Fanuc KAREL source: kt00452.KL

-- PROVISIONAL review KL for V770-1; original PC SHA256 5246766105a77e096c1f6754eb6137f0ccf5cd3cca0d1063bb0bf1915763c5d0
-- Incomplete behavior may be omitted. Consult companion uncertainty JSON. Do not deploy.
PROGRAM KT00452
%NOLOCKGROUP
VAR
  R2 : REAL
  OUT : BOOLEAN
-- UNRESOLVED_DECL H1 type=002017
BEGIN
  -- UNRESOLVED_PC offsets 5-19; opcodes 2E,22,9D,33,B4
  -- UNRESOLVED_PC offsets 24-35; opcodes 2E,23
  -- UNRESOLVED_PC offsets 40-65; opcodes 22,9D,33,B3,21,29,64,29,72,23
  -- UNRESOLVED_PC offsets 70-74; opcodes 7F
END KT00452
